FUNCTION_BLOCK DisableGroup  IMPLEMENTS I_Task
VAR
	groupDisable		: MC_GroupDisable;
	_caGroup			: I_CollisionGroup;
	_Done 				: BOOL;
	_Error				: BOOL;
	_ErrorID			: UDINT;
END_VAR

{analysis -2}

METHOD Abort : BOOL
groupDisable.Execute := FALSE;
Abort := true;
END_METHOD

PROPERTY Busy : BOOL
GET
Busy := groupDisable.Busy;
END_GET
END_PROPERTY

METHOD Cycle : HRESULT
VAR_INPUT
END_VAR
IF _caGroup = 0 THEN
	cycle := -1;
	RETURN;
END_IF
_Done := groupDisable.Done OR _Done;
_Error := groupDisable.Error OR _Error;
IF groupDisable.ErrorId <> 0 THEN
	_ErrorId := groupDisable.ErrorId;
END_IF
groupDisable(AxesGroup := _caGroup.GroupRef);
groupDisable.Execute := false;
END_METHOD

PROPERTY Done : BOOL
GET
Done := _Done;
END_GET
END_PROPERTY

PROPERTY Error : BOOL
GET
Error := _Error;
END_GET
END_PROPERTY

METHOD Execute : hresult
IF groupDisable.Execute THEN
	Execute := -1;
	RETURN;
END_IF

IF _caGroup = 0 THEN
	Execute := -2;
	RETURN;
END_IF
groupDisable.Execute := TRUE;
END_METHOD

PROPERTY MyCollisionGroup : I_CollisionGroup
GET
MyCollisionGroup := _caGroup;
END_GET
SET
IF MyCollisionGroup <> 0 THEN
	_caGroup := MyCollisionGroup;
END_IF
END_SET
END_PROPERTY

END_FUNCTION_BLOCK

(* stored: Version 1.1.0.1
   POU DisableGroup: Id {e309beac-a8f6-4753-8ed9-d8f37883f7b3}, SpecialFunc None
   Method Abort: Id {471c738d-2cd1-4d5e-b4b6-abdacd440e10}
   Property Busy: Id {32df597f-701e-4887-9694-05ec5ec7d053}
   Get Get: Id {bc9c2786-f3ce-4ee5-a9c4-8b58d5ce6f43}
   Method Cycle: Id {8091e283-75fa-4fa7-b8ef-612c591a9cfd}
   Property Done: Id {6399d63a-c4a7-4051-98bb-74ddbb9f8698}
   Get Get: Id {6f70f022-3ee9-4c34-a58e-db5d8234b980}
   Property Error: Id {1bd1c661-8257-4434-b6a5-6f6723f1e85f}
   Get Get: Id {4115ab3f-61e6-4ab9-b302-760db309b763}
   Method Execute: Id {957a3466-1261-44df-92f7-84f5463a1c53}
   Property MyCollisionGroup: Id {374f3446-8902-46b9-be62-e00e0857d034}
   Get Get: Id {1f6f12f3-f514-420f-acb0-8e57d892b9eb}
   Set Set: Id {3ccd05ee-eb7b-4371-a968-95a0571a1e90} *)
